TYPE "ST_HmiResponse"
VERSION : 0.1
   STRUCT
      AckSequence : UDInt;
      Accepted : Bool;
      Diagnostic : String[64];     // localization key when refused
   END_STRUCT;

END_TYPE
